FUNCTION_BLOCK SAFE_DAC_RATE_LIMITER (* DAC rate limiter with deterministic startup, reset, bounds, and diagnostics *)
  (* Standard: 61499-2 *)
  (* Version 1.0, 2026-07-26, Guilherme *)
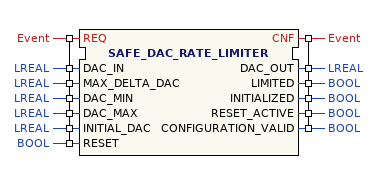
  EVENT_INPUT
    REQ WITH DAC_IN, MAX_DELTA_DAC, DAC_MIN, DAC_MAX, INITIAL_DAC, RESET; (* Execute one safe DAC rate-limiter cycle *)
  END_EVENT
  EVENT_OUTPUT
    CNF WITH DAC_OUT, LIMITED, INITIALIZED, RESET_ACTIVE, CONFIGURATION_VALID; (* Safe DAC rate-limiter cycle completed *)
  END_EVENT
  VAR_INPUT
    DAC_IN : LREAL; (* Requested DAC command *)
    MAX_DELTA_DAC : LREAL; (* Maximum DAC output change per execution *)
    DAC_MIN : LREAL; (* Minimum allowed DAC output *)
    DAC_MAX : LREAL; (* Maximum allowed DAC output *)
    INITIAL_DAC : LREAL; (* Deterministic output used at startup and reset *)
    RESET : BOOL; (* Apply deterministic reset behavior *)
  END_VAR
  VAR_OUTPUT
    DAC_OUT : LREAL; (* Bounded and rate-limited DAC output *)
    LIMITED : BOOL; (* Output differs from the requested DAC input *)
    INITIALIZED : BOOL; (* Limiter has valid initialized state *)
    RESET_ACTIVE : BOOL; (* Current cycle executed reset behavior *)
    CONFIGURATION_VALID : BOOL; (* Rate and output-limit configuration is valid *)
  END_VAR
  VAR
    previous_dac : LREAL := 0.0; (* Stored DAC output from the previous valid cycle *)
    initialized_internal : BOOL := FALSE; (* Internal initialization state *)
    bounded_input : LREAL := 0.0; (* Requested DAC after output bounds *)
    bounded_initial : LREAL := 0.0; (* Initial DAC after output bounds *)
    delta_dac : LREAL := 0.0; (* Difference between bounded input and previous output *)
    limited_delta : LREAL := 0.0; (* DAC difference after rate limiting *)
  END_VAR
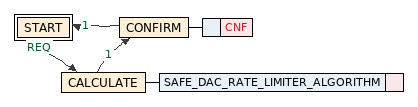
  EC_STATES
    START; (* Initial state *)
    CALCULATE : SAFE_DAC_RATE_LIMITER_ALGORITHM; (* Execute safe DAC rate limiting *)
    CONFIRM : -> CNF; (* Publish limiter outputs *)
  END_STATES
  EC_TRANSITIONS
    START TO CALCULATE := REQ;
    CALCULATE TO CONFIRM := 1;
    CONFIRM TO START := 1;
  END_TRANSITIONS
  ALGORITHM SAFE_DAC_RATE_LIMITER_ALGORITHM IN ST: (* Deterministic startup, reset, bounds, and symmetric DAC rate limiting *)
CONFIGURATION_VALID :=
    (MAX_DELTA_DAC > 0.0)
    AND
    (DAC_MIN < DAC_MAX);

IF NOT CONFIGURATION_VALID THEN
    previous_dac := 0.0;
    initialized_internal := FALSE;

    DAC_OUT := 0.0;
    LIMITED := TRUE;
    INITIALIZED := FALSE;
    RESET_ACTIVE := FALSE;

ELSE
    bounded_initial := INITIAL_DAC;

    IF bounded_initial > DAC_MAX THEN
        bounded_initial := DAC_MAX;
    ELSIF bounded_initial < DAC_MIN THEN
        bounded_initial := DAC_MIN;
    END_IF;

    IF RESET OR NOT initialized_internal THEN
        previous_dac := bounded_initial;
        DAC_OUT := previous_dac;
        initialized_internal := TRUE;

        LIMITED := DAC_OUT <> DAC_IN;
        INITIALIZED := TRUE;
        RESET_ACTIVE := RESET;

    ELSE
        bounded_input := DAC_IN;

        IF bounded_input > DAC_MAX THEN
            bounded_input := DAC_MAX;
        ELSIF bounded_input < DAC_MIN THEN
            bounded_input := DAC_MIN;
        END_IF;

        delta_dac := bounded_input - previous_dac;

        IF delta_dac > MAX_DELTA_DAC THEN
            limited_delta := MAX_DELTA_DAC;
        ELSIF delta_dac < -MAX_DELTA_DAC THEN
            limited_delta := -MAX_DELTA_DAC;
        ELSE
            limited_delta := delta_dac;
        END_IF;

        DAC_OUT := previous_dac + limited_delta;

        IF DAC_OUT > DAC_MAX THEN
            DAC_OUT := DAC_MAX;
        ELSIF DAC_OUT < DAC_MIN THEN
            DAC_OUT := DAC_MIN;
        END_IF;

        previous_dac := DAC_OUT;

        LIMITED := DAC_OUT <> DAC_IN;
        INITIALIZED := TRUE;
        RESET_ACTIVE := FALSE;
    END_IF;
END_IF;
  END_ALGORITHM
END_FUNCTION_BLOCK
